FUNCTION_BLOCK FB_SuctionCup_Sim IMPLEMENTS I_SuctionCup
VAR_INPUT
END_VAR
VAR_OUTPUT
END_VAR
VAR
	fPressure 			: REAL;// Value 0-100 %
	bSuck				: BOOL;
	// var sim
	tTimer				: TON;
	tDelay				: TIME := T#1000MS;// acceleration time of fPressure to value = 100
	nState				: INT := 0;
	bRelease			: BOOL := TRUE;
END_VAR

CASE nState OF
	0: //init release Suction
		IF bRelease THEN
			bSuck := FALSE;
			fPressure := 0;
		ELSE
			bSuck := TRUE;
			fPressure := 100;
		END_IF
		tTimer(IN := FALSE);
		nState := nState + 1;
	1:// check for signal
		tTimer(IN := FALSE);
		IF bSuck AND (fPressure = 0) THEN
			nState := 10;
		END_IF
		IF NOT bSuck AND (fPressure = 100) THEN
			nState := 20;
		END_IF
	10: //Suck 
		tTimer(IN := TRUE,PT := tDelay);
		fPressure := TIME_TO_REAL(tTimer.ET)*(100/TIME_TO_REAL(tDelay));
		IF (fPressure = 100) THEN
			nState := 1;
		END_IF
	20:// release
		tTimer(IN := TRUE,PT := tDelay);
		fPressure := 100 - (TIME_TO_REAL(tTimer.ET)*(100/TIME_TO_REAL(tDelay)));
		IF (fPressure = 0) THEN
			nState := 1;
		END_IF
END_CASE

PROPERTY bIsSuck : BOOL
GET
IF fPressure > fThreshold THEN
	bIsSuck := TRUE;
ELSE 
	bIsSuck := FALSE;
END_IF
END_GET
END_PROPERTY

PROPERTY fThreshold : REAL
GET
fThreshold := 50;
END_GET
SET
END_SET
END_PROPERTY

METHOD Release : BOOL
VAR_INPUT
END_VAR
bSuck := FALSE;
END_METHOD

METHOD Suck : BOOL
VAR_INPUT
END_VAR
bSuck := TRUE;
END_METHOD

END_FUNCTION_BLOCK

(* stored: Version 1.1.0.1, ProductVersion 3.1.4024.12
   POU FB_SuctionCup_Sim: Id {66b54f8e-cd6e-49f1-a63b-0d9b3ba7cb64}, SpecialFunc None
   Property bIsSuck: Id {413d8c2a-4fc7-4c33-b68c-d7fed262ced3}
   Get Get: Id {ed8cbd51-05d0-4216-9cae-eeea3ad4fadc}
   Property fThreshold: Id {54931e21-7f12-4014-8004-1dcda19fe3c8}
   Get Get: Id {5b8425b8-304a-4ec8-9797-5606ac7d58fa}
   Set Set: Id {45cc4d9c-453c-47a4-bec2-113bb997aa4f}
   Method Release: Id {8461aea9-1726-4a5e-aa5b-8dbf45b93a5f}
   Method Suck: Id {1da0afd0-7312-49b8-916e-5a4f627ce6d7} *)
